// TIA Portal V18 export
TYPE "UDT_AHUEqpDemand"
// stored: IsFailsafeCompliant false
   STRUCT
      rFan : Array[1..3] of Real;   // 0-wout ctrl/1 - ProxiAdaptation/
      rExtractDumper : Array[1..3] of Real;   // 0-wout ctrl/1 - ProxiAdaptation/
      rMixingDumper : Array[1..3] of Real;   // 0-wout ctrl/1 - ProxiAdaptation/
      rHeater : Array[1..3] of Real;   // 0-wout ctrl/1 - ProxiAdaptation/
      rCooler : Array[1..3] of Real;   // 0-wout ctrl/1 - ProxiAdaptation/
      rWHU : Array[1..3] of Real;   // 0-wout ctrl/1 - ProxiAdaptation/
   END_STRUCT;
END_TYPE
